// TIA Portal project "Project" (V17)

(* hardware
DEVICE "S7-300/ET200M station_1"  S7-300 station
   slot 0: "Rail_0"  Rail  6ES7 390-1***0-0AA0
   slot 2: "PLC_1"  CPU 315-2 PN/DP  6ES7 315-2EH13-0AB0  V2.6
      slot 1: "MPI/DP interface_1"  X1
      slot 2: "PROFINET interface_1"  PN-IO
         slot 1: "Port_1"  Port
   slot 4: "AI 4x0/4mA/20mA, Ex_1"  AI4 x 0/4 to 20mA, Ex  6ES7 331-7RD00-0AB0
   slot 5: "AO 4x0/4..20mA, Ex_1"  AO4 x 0/4 to 20mA, Ex  6ES7 332-5RD00-0AB0
   slot 6: "DI 32x24VDC_1"  DI32 x 24VDC  6ES7 321-1BL00-0AA0
   slot 7: "DO 32x24VDC/0.5A_1"  DO32 x 24VDC / 0.5A  6ES7 322-1BL00-0AA0
DEVICE "PSU8600 station_1"  PSU8600 station
   slot 0: "Rack_0"  Rail
   slot 0: "PSU_1"  PSU8600 1ph 20A/4x5A PN  6EP3336-8MB00-2CY0  V1.5
DEVICE "HMI_1"  KTP700 Basic DP
   slot 0: "HMI_1"  KTP700 Basic DP  6AV2 123-2GA03-0AX0  17.0.0.0
   slot 1: "HMI_RT_1"  KTP700 Basic DP  6AV2 123-2GA03-0AX0  17.0.0.0
   slot 7: "HMI_1.MPI/DP_CP_1"  MPI/DP Interface  17.0.0.0
*)

// ===== PLC "PLC_1"  CPU 315-2 PN/DP =====

VAR_GLOBAL   // PLC tag table "Default tag table"
   "STOP" AT %I0.0 : Bool;
   "START" AT %I0.1 : Bool;
   "HEATER_PREHEAT" AT %M0.0 : Bool;
   "COUNT" AT %MW2 : Int;
   "MIXER" AT %M0.1 : Bool;
   "OPEN_PUMP" AT %I0.2 : Bool;
   "CLOSE_PUMP" AT %I0.3 : Bool;
   "POSITION" AT %MW4 : Int;
   "FILTER_UNIT" AT %M0.2 : Bool;
END_VAR

ORGANIZATION_BLOCK "Main"   // OB1, LAD
TITLE = "Main Program Sweep (Cycle)"
{ S7_Optimized_Access := 'FALSE' }
VERSION : 0.1
   VAR_TEMP
      OB1_EV_CLASS : Byte;   // Bits 0-3 = 1 (Coming event), Bits 4-7 = 1 (Event class 1)
      OB1_SCAN_1 : Byte;   // 1 (Cold restart scan 1 of OB 1), 3 (Scan 2-n of OB 1)
      OB1_PRIORITY : Byte;   // Priority of OB Execution
      OB1_OB_NUMBR : Byte;   // 1 (Organization block 1, OB1)
      OB1_RESERVED_1 : Byte;   // Reserved for system
      OB1_RESERVED_2 : Byte;   // Reserved for system
      OB1_PREV_CYCLE : Int;   // Cycle time of previous OB1 scan (milliseconds)
      OB1_MIN_CYCLE : Int;   // Minimum cycle time of OB1 (milliseconds)
      OB1_MAX_CYCLE : Int;   // Maximum cycle time of OB1 (milliseconds)
      OB1_DATE_TIME : Date_And_Time;   // Date and time OB1 started
   END_VAR
BEGIN

REGION Network 1
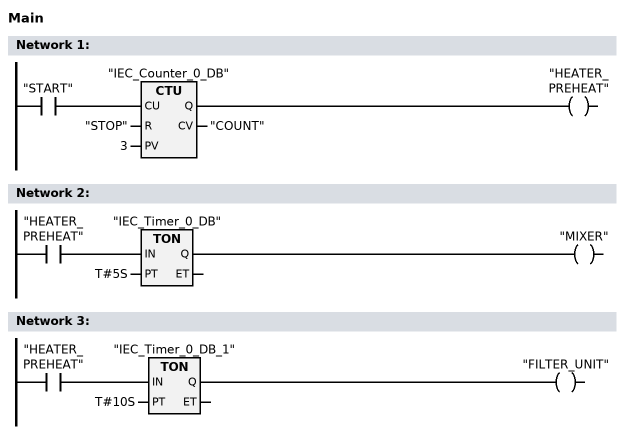
   "IEC_Counter_0_DB".CTU(CU := "START", R := "STOP", PV := 3, CV => "COUNT");
   "HEATER_PREHEAT" := "IEC_Counter_0_DB".Q;
END_REGION

REGION Network 2
   "IEC_Timer_0_DB".TON(IN := "HEATER_PREHEAT", PT := T#5S);
   "MIXER" := "IEC_Timer_0_DB".Q;
END_REGION

REGION Network 3
   "IEC_Timer_0_DB_1".TON(IN := "HEATER_PREHEAT", PT := T#10S);
   "FILTER_UNIT" := "IEC_Timer_0_DB_1".Q;
END_REGION
END_ORGANIZATION_BLOCK

ORGANIZATION_BLOCK "CYC_INT5"   // OB35, LAD
TITLE = "Cyclic Interrupt"
{ S7_Optimized_Access := 'FALSE' }
VERSION : 0.1
   VAR_TEMP
      OB35_EV_CLASS : Byte;   // Bits 0-3 = 1 (Coming event), Bits 4-7 = 1 (Event class 1)
      OB35_STRT_INF : Byte;   // 16#36 (OB 35 has started)
      OB35_PRIORITY : Byte;   // Priority of OB Execution
      OB35_OB_NUMBR : Byte;   // 35 (Organization block 35, OB35)
      OB35_RESERVED_1 : Byte;   // Reserved for system
      OB35_RESERVED_2 : Byte;   // Reserved for system
      OB35_PHASE_OFFSET : Word;   // Phase offset (msec)
      OB35_RESERVED_3 : Int;   // Reserved for system
      OB35_EXC_FREQ : Int;   // Frequency of execution (msec)
      OB35_DATE_TIME : Date_And_Time;   // Date and time OB35 started
   END_VAR
BEGIN

REGION Network 1
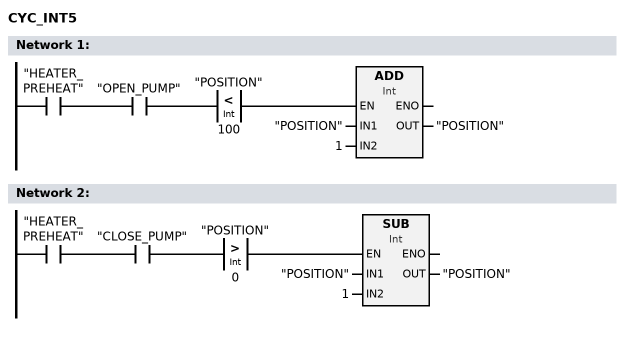
   RUNG wire#powerrail
      Contact( "HEATER_PREHEAT" )
      Contact( "OPEN_PUMP" )
      { S7_Templates := "SrcType := Int" } LT_Contact(in1 := "POSITION", in2 := 100)
      { S7_Templates := "SrcType := Int"; S7_GenerateENO := "TRUE" } Add(in1 := "POSITION", in2 := 1, out => "POSITION")
   END_RUNG
   // the same network as SCL:
   IF "HEATER_PREHEAT" AND "OPEN_PUMP" AND ("POSITION" < 100) THEN "POSITION" := "POSITION" + 1; END_IF;
END_REGION

REGION Network 2
   RUNG wire#powerrail
      Contact( "HEATER_PREHEAT" )
      Contact( "CLOSE_PUMP" )
      { S7_Templates := "SrcType := Int" } GT_Contact(in1 := "POSITION", in2 := 0)
      { S7_Templates := "SrcType := Int"; S7_GenerateENO := "TRUE" } Sub(in1 := "POSITION", in2 := 1, out => "POSITION")
   END_RUNG
   // the same network as SCL:
   IF "HEATER_PREHEAT" AND "CLOSE_PUMP" AND ("POSITION" > 0) THEN "POSITION" := "POSITION" - 1; END_IF;
END_REGION
END_ORGANIZATION_BLOCK

(* ===== HMI "HMI_RT_1" =====
system functions are stored by id; their names below are inferred from use
connection "HMI_Connection_1": IF1 B, SIMATIC S7 300/400 MPI

HMI tags "Default tag table"
   "Tag_ScreenNumber" : UInt, internal
   "STOP" : Bool = PLC STOP AT %I0.0, 1 s
   "START" : Bool = PLC START AT %I0.1, 1 s
   "HEATER_PREHEAT" : Bool = PLC HEATER_PREHEAT AT %M0.0, 1 s
   "MIXER" : Bool = PLC MIXER AT %M0.1, 1 s
   "OPEN_PUMP" : Bool = PLC OPEN_PUMP AT %I0.2, 1 s
   "CLOSE_PUMP" : Bool = PLC CLOSE_PUMP AT %I0.3, 1 s
   "POSITION" : Int = PLC POSITION AT %MW4, 1 s
   "FILTER_UNIT" : Bool = PLC FILTER_UNIT AT %M0.2, 1 s

Template "Template_1" 800x480
   Button "Exit" at 714,429 size 71x50; TextOff 'Exit'; PictureOff "ExitRuntime_KTP700_Basic_DP_TR"; PictureOn "ExitRuntime_KTP700_Basic_DP_TR"
      on Release: StopRuntime(0)
   Button "Template_Button" at 614,429 size 71x50; TextOff 'Text'
   Button "Template_Button_1" at 514,429 size 71x50; TextOff 'Text'
   Button "Template_Button_2" at 414,429 size 71x50; TextOff 'Text'
   Button "Template_Button_3" at 314,429 size 71x50; TextOff 'Text'
   Button "Template_Button_4" at 214,429 size 71x50; TextOff 'Text'
   Button "Template_Button_5" at 114,429 size 71x50; TextOff 'Text'
   Button "Start screen" at 14,429 size 71x50; TextOff 'Start screen'; PictureOff "NavigateHome_KTP700_Basic_DP_TR"; PictureOn "NavigateHome_KTP700_Basic_DP_TR"
      on Release: ActivateScreen("Root screen", 0)
   SymbolicIOField "Symbolic_IO_Field_Screen" at 93,9 size 600x33; TextOff '0'; TextOn '1'; TextList "TextList_ScreenNames"
      ProcessValue <- "Tag_ScreenNumber"
      on Change: ActivateScreenByNumber("Tag_ScreenNumber", 0)
   DateTimeField "HmiScreenItemData" at 695,25 size 105x25
   DateTimeField "HmiScreenItemData_1" at 695,0 size 105x25
   GraphicView "Logo" at 0,0 size 91x51; Picture "Logo of HMI_1"

screen "Root screen" 800x480, template "Template_1"
   on GenerateScreen: SetTag("Tag_ScreenNumber", 1)
   TextField "Text field_1" at 218,63 size 352x28; Text 'Предварительная очистка нефти'
   Button "Button_1" at 16,106 size 122x122; TextOff 'Старт'
      on Press: SetBit("START")
      on Release: ResetBit("START")
   Button "Button_2" at 150,106 size 122x122; TextOff 'Стоп'
      on Press: SetBit("STOP"); SetTag("POSITION", 0)
      on Release: ResetBit("STOP")
   Circle "Circle_1" at 22,244 size 48x48
      Appearance <- "HEATER_PREHEAT"
   TextField "Text field_2" at 80,255 size 65x23; Text 'Нагрев'
   Circle "Circle_2" at 22,303 size 48x48
      Appearance <- "MIXER"
   TextField "Text field_3" at 80,314 size 84x23; Text 'Мешалка'
   Circle "Circle_3" at 22,360 size 48x48
      Appearance <- "FILTER_UNIT"
   TextField "Text field_4" at 80,371 size 107x23; Text 'Фильтрация'
   TextField "Text field_5" at 612,106 size 91x23; Text 'Задвижка'
   IOField "I/O field_1" at 612,133 size 96x32; FormatPattern s999
      ProcessValue <- "POSITION"
   Button "Button_3" at 535,182 size 96x32; TextOff 'Открыть'
      on Press: SetBit("OPEN_PUMP")
      on Release: ResetBit("OPEN_PUMP")
   Button "Button_4" at 683,182 size 96x32; TextOff 'Закрыть'
      on Press: SetBit("CLOSE_PUMP")
      on Release: ResetBit("CLOSE_PUMP")
*)